{attribute 'GeneratedUsingTerminal: EJ9576-0000-0020'}
{attribute addProperty BoxType "EJ9576-0000-0020"}
{attribute addProperty Id "EtcSlaveTerminalBaseBCT_InputsAT %I*BCT_Inputs_8B1D510C16WcStateAT %I*WcState_9091E0EB2InfoDataAT %I*InfoData_32EB74EA10"}
{attribute addProperty CRC "305678668"}
{attribute addProperty Size "28"}
TYPE EJ9576_1238494C EXTENDS EtcSlaveTerminalBase :
STRUCT
	{attribute addProperty Name "BCT_Inputs"}
	BCT_Inputs : BCT_Inputs_8B1D510C;
	{attribute addProperty Name "WcState"}
	WcState : WcState_9091E0EB;
	{attribute addProperty Name "InfoData"}
	InfoData : InfoData_32EB74EA;
END_STRUCT
END_TYPE

(* stored: Version 1.2.0.0, ProductVersion 3.1.4024.9
   DUT EJ9576_1238494C: Id {a4e4427b-8a45-4266-ba78-6535317cb429} *)
